INTERFACE ITF_EM_Transport_StampUnit_SealShrink

END_INTERFACE

(* stored: Version 1.1.0.1, ProductVersion 3.1.4024.12
   Itf ITF_EM_Transport_StampUnit_SealShrink: Id {7c18349a-38d6-425e-a306-2fe202877357} *)
